Staubli VAL3: RefreshList.pgx

program RefreshList()
  local num l_ni
begin
  if bListRefresh
    resize(sList,1,size(pPoint))
    for l_ni=0 to size(pPoint)-1
      sList[l_ni]="P"+toString("",l_ni+1)
    endFor
  endIf
end
